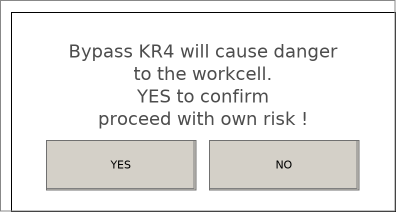
VISUALIZATION MSG_KR3_BP  // 396x212
    RoundedRectangle (11,12 385x200)
    Button (46,140 150x50), "YES"
        OnMouseClick: CloseDialog Dialog=MSG_KR3_BP, Result=Yes, NumpadKeypadSet=True
        OnMouseClick: execute { GVL.KR3_bypass := TRUE; }
    Button (209,140 150x50), "NO"
        OnMouseClick: execute { GVL.KR3_bypass := FALSE; }
        OnMouseClick: CloseDialog Dialog=MSG_KR3_BP, Result=No, NumpadKeypadSet=True
    Label (55,30 296x110), "Bypass KR4 will cause danger to the workcell. YES to confirm proceed with own risk !"
END_VISUALIZATION

(* stored: Version 1.1.0.1, ProductVersion 3.1.4024.12
   Visu MSG_KR3_BP: Id {555f2061-be7d-48e6-896b-aa23fd5fa0cd} *)
